// TwinCAT 3 PLC project HttpRequest
// ProgramVersion: 3.1.4024.0
// libraries:
//   Tc2_Standard, * (Beckhoff Automation GmbH)
//   Tc2_System, * (Beckhoff Automation GmbH)
//   Tc2_Utilities, * (Beckhoff Automation GmbH)
//   Tc3_IotBase, * (Beckhoff Automation GmbH)
//   Tc3_JsonXml, * (Beckhoff Automation GmbH)
//   Tc3_Module, * (Beckhoff Automation GmbH)
// project tree:
//   / PlcTask.TcTTO
//   POUs/HTTP/ FB_EventHTTP_Post.TcPOU
//   POUs/ MAIN.TcPOU
// real-time tasks:
//   TASK PlcTask: cycle T#10ms, priority 20, ADS port 350
// I/O:
//   DEVICE Device 1 (EtherCAT) (disabled), AmsNetId 192.168.1.132.2.1
//     Term 1 (EK1100) [EK1100 EtherCAT Coupler (2A E-Bus)]
//       Term 2 (EL1889) [EL1889 16Ch. Dig. Input 24V, 3ms, negative]
//       Term 3 (EL2889) [EL2889 16Ch. Dig. Output 24V, 0.5A, negative]
//       Term 4 (EL9011) [EL9011 End Terminal]

CONFIGURATION HttpRequest
    RESOURCE PLC ON TwinCAT3
        TASK PlcTask(INTERVAL := T#10ms, PRIORITY := 20);
        PROGRAM MAIN WITH PlcTask : MAIN;
    END_RESOURCE
END_CONFIGURATION

// ---- POUs/MAIN.TcPOU
PROGRAM MAIN
VAR
	IPAdress		: STRING 	:= '192.168.1.168';
	Port			: UINT		:= 8080;
	UpdatePeriod	: TIME		:= T#60s;
	fbHttpProcess	: FB_IotHttpClient :=(	sHostName			:= IPAdress,
								  			bKeepAlive			:= TRUE, 
											tConnectionTimeout	:= T#10S);
	fbProcessPost	: FB_EventHTTP_Post;
	
	HttpSend		: BOOL := FALSE;
	
	API_Msg			: STRING[255] := '';
	bSuccess		: BOOL;
	bError			: BOOL;
END_VAR


IF NOT fbHttpProcess.bConfigured THEN 
	fbHttpProcess.nHostPort 				:= Port;
	fbHttpProcess.stTLS.bNoServerCertCheck 	:= TRUE;
END_IF

IF fbHttpProcess.bConfigured THEN 
	fbProcessPost( 	bSend		:= HttpSend, 
				 	fbClient	:= fbHttpProcess, 
					API_URI		:= '/Workcell_Logging',
				 	API_Msg 	:= API_Msg,
					bSuccess 	=> bSuccess,
					bError		=> bError );
END_IF 
fbHttpProcess.Execute();

END_PROGRAM

// ---- POUs/HTTP/FB_EventHTTP_Post.TcPOU
FUNCTION_BLOCK FB_EventHTTP_Post
VAR_INPUT
	bSend		: BOOL;
	API_URI		: STRING[255];
	API_Msg		: STRING[255];
END_VAR
VAR_IN_OUT
	fbClient			: FB_IotHttpClient;
END_VAR
VAR_OUTPUT
	bSuccess			: Bool;
	bBusy				: BOOL;
	bError				: BOOL;
END_VAR
VAR	
	fbRequest			: FB_IotHttpRequest;
	fbJson				: FB_JsonDomParser;
	
 	dtTimestamp    		: DATE_AND_TIME := DT#2017-04-04-12:42:42;
	fbJsonWriter		: FB_JsonDomParser;
	nState				: UDINT;
	RisingEdge			: R_TRIG;
	
	bGetContentResult	: BOOL;
	sContent			: STRING[255] := ''; 
	
	bGetJsonResult		: BOOL;
	jsonDoc				: SJsonValue;
	jsonVal				: SJsonValue;
	sResultValue		: STRING;
	
	nReqCount			: UDINT;
	nResCount			: UDINT;
	nValidResCount		: UDINT;
	nErrCount			: UDINT;	
END_VAR

RisingEdge(CLK:= bSend);
CASE nState OF
0:		
	IF RisingEdge.Q THEN 
		sContent := API_Msg;		
		IF fbRequest.SendRequest(sUri:= API_URI, fbClient:= fbClient, eRequestType:= ETcIotHttpRequestType.HTTP_POST, pContent:= ADR(sContent), nContentSize:= LEN2(ADR(sContent)), 0) THEN				
			nState:= 1;
			bBusy:= TRUE;
			bError:= FALSE;
			bSuccess := FALSE;
		END_IF					
	END_IF
1:
	IF NOT fbRequest.bBusy THEN
		bError:= TRUE;
		IF NOT fbRequest.bError THEN				 				
			bGetContentResult:= fbRequest.GetContent(pContent:= ADR(sContent), nContentSize:= SIZEOF(SContent), bSetNullTermination:= TRUE);	
			IF fbRequest.nStatusCode >= 200 AND fbRequest.nStatusCode < 300 THEN
				bGetJsonResult:= FALSE;
				jsonDoc:= fbRequest.GetJsonDomContent(fbJson);				
				IF jsonDoc <> 0 THEN
					bGetJsonResult:= TRUE;
					IF fbJson.HasMember(jsonDoc, 'status')  THEN
						jsonVal:= fbJson.FindMember(jsonDoc, 'status');
						sResultValue:= fbJson.GetString(jsonVal);
						IF sResultValue = 'success' THEN
							nValidResCount:= nValidResCount+1;
							bSuccess := TRUE;//////////////////////////////////////////////////
							bError:= FALSE;
						END_IF
					END_IF		
				END_IF
				nResCount:= nResCount+1;					
			END_IF				
		END_IF
		nState:= 0;
		bBusy:= FALSE;
		IF bError THEN
			nErrCount:= nErrCount+1;
		END_IF		
	END_IF 
END_CASE

END_FUNCTION_BLOCK
